TYPE ST_UN_Machine100_Cmd :
STRUCT
	bCmdRun			: BOOL;
	bCmdRunEmpty	: BOOL;
	
END_STRUCT
END_TYPE

(* stored: Version 1.1.0.1, ProductVersion 3.1.4024.10
   DUT ST_UN_Machine100_Cmd: Id {d2f2fdb2-77f3-4cc2-b111-15048e201c43} *)
